FUNCTION rt_remd : LREAL
VAR_INPUT
	u0: LREAL;
	u1: LREAL;
END_VAR
VAR
	u: LREAL;
	tmp: LREAL;
END_VAR


u := u0 / u1;

IF u1 <= rt_floord(u := u1) THEN 
    rt_remd := u0 - (DINT_TO_LREAL(TRUNC(u)) * u1);
ELSE 
    tmp := ABS(u);

    IF tmp < 4.503599627370496E+15 THEN 

        IF u >= 0.5 THEN 
            rt_remd := rt_floord(u := u + 0.5);
        ELSIF u > -0.5 THEN 
            rt_remd := 0.0;
        ELSE 
            rt_remd := rt_ceild(u := u - 0.5);
        END_IF;

    ELSE 
        rt_remd := u;
    END_IF;


    IF ABS(u - rt_remd) <= (2.2204460492503131E-16 * tmp) THEN 
        rt_remd := 0.0;
    ELSE 
        rt_remd := (u - DINT_TO_LREAL(TRUNC(u))) * u1;
    END_IF;

END_IF;

END_FUNCTION

(* stored: Version 1.1.0.1, ProductVersion 3.1.4024.12
   POU rt_remd: Id {8df6122e-14d1-4160-94f0-b83dde04e87b}, SpecialFunc None *)
